ABB RAPID module: CalibData.modx

MODULE CalibData
	PERS wobjdata TABLE1 := [FALSE,TRUE,"",[[734.0569,628.4146,766.7589],[0.9657609,-0.005640136,-0.2593307,-0.004649641]],[[0,0,0],[1,0,0,0]]];
	PERS wobjdata TABLE2 := [FALSE,TRUE,"",[[0,0,0],[1,0,0,0]],[[0,0,0],[1,0,0,0]]];
ENDMODULE
